INTERFACE I_BothMovers EXTENDS I_SingleMover

PROPERTY Mover2 : I_XPlanarMover
GET
END_GET
SET
END_SET
END_PROPERTY

END_INTERFACE

(* stored: Version 1.1.0.1, ProductVersion 3.1.4026.20
   Itf I_BothMovers: Id {210507a2-603b-49d4-88c1-4d5d176a9a0c}
   Property Mover2: Id {8ea4ab8c-3229-41cb-b6e1-f0575bc1fa47}
   Get Get: Id {30d8c4f8-ad99-421c-8dde-2400d088f962}
   Set Set: Id {9b482b1a-7bc6-475c-800b-beb0dd0b1cf8} *)
